// TIA Portal V16 export
// export: Created 2023-03-29T11:05:06.0398935Z, ExportSetting WithDefaults, DisplayName Totally Integrated Automation Portal, DisplayVersion V16 Update 6, DisplayName TIA Portal Version Control Interface, DisplayVersion V16 Update 2, DisplayName TIA Portal Openness, DisplayVersion V16 Update 6, DisplayName STEP 7 Professional, DisplayVersion V16 Update 6, DisplayName STEP 7 Safety, DisplayVersion V16, DisplayName WinCC Advanced, DisplayVersion V16 Update 6
VAR_GLOBAL   // PLC tag table "Error"
   Led_Error AT %M17.5 : Bool;   // Znacznik sygnalizujący wystąpienie błędu sterownika Krat
   ResetErrorOB82 AT %M17.4 : Bool;   // Znacznik resetu licznika błędów
   alarmSuchobieg AT %M93.2 : Bool;   // bit alarmu wystąpienia suchobiegu pompownia
   alarmMagistrala_niskie_bar AT %M93.3 : Bool;   // bit alarmu wystąpienia btraku ciśnienia z magistrali
   "off_AlarmMagistrala-niskie_bar" AT %M93.4 : Bool;   // bit informuje o końcu awarii magistrali niskie
   alarm_max_bar_pompownia AT %M94.0 : Bool;   // bit alarmu przekroczono max bar pompownia B7
   Discrete_alarm_18 AT %M1025.1 : Bool;   // 16#0002: Niepoprawna wartość w parametrze "Input_PER". Sprawdź, czy na wejściu analogowym występuje błąd.
   "BitMeldun-7" AT %M1029.7 : Bool;   // 16#0080: Niepoprawna wartość w trybie pracy PID. Tryb pracy nie ulega zmianie.
   Discrete_alarm_13 AT %M1024.4 : Bool;   // 16#1000: Niepoprawna wartość w parametrze "Wartość zadana": Wartość nie ma prawidłowego formatu liczbowego.
   tmp_rezerwa_1 AT %M94.1 : Bool;   // bit rezerwowy 1
   bit_off_alarm_magistrala AT %M94.2 : Bool;   // ustaw jesli koniec alarmu na magistrali bar <min
END_VAR
